Staubli VAL3: save.pgx

public program save(num& x_nResult[])
  local num i
begin
  x_nResult=saveData:libSave()
end
